(* IEC 61131-3 sources: AXOpen/src/components.abb.robotics/ctrl/src/AxoIrc5_v_1_x_x/TypesStructuresAndEnums, 5 files *)

(* ---- AxoIrc5_v_1_x_x_Component_Status.st ---- *)
NAMESPACE AXOpen.Components.Abb.Robotics
    {S7.extern=ReadWrite}
    {#ix-attr:[Container(Layout.Stack)]}
    CLASS PUBLIC AxoIrc5_v_1_x_x_Component_Status  EXTENDS AXOpen.Components.Robotics.AxoRobot_Status
        VAR PUBLIC
        END_VAR
    END_CLASS
END_NAMESPACE

(* ---- AxoIrc5_v_1_x_x_Config.st ---- *)
NAMESPACE AXOpen.Components.Abb.Robotics
    {#ix-attr:[Container(Layout.Stack)]}
    {S7.extern=ReadWrite}
    CLASS PUBLIC AxoIrc5_v_1_x_x_Config
        VAR PUBLIC
            {#ix-set:AttributeName = "<#Info time#>"}
            InfoTime : LTIME := LT#2S;
            {#ix-set:AttributeName = "<#Error time#>"}
            ErrorTime : LTIME := LT#0S;
            {#ix-set:AttributeName = "<#Task timeout#>"}
            TaskTimeout : LTIME := LT#0S;
            {#ix-set:AttributeName = "<#Hardware IDs#>"}
            HWIDs : AxoIrc5_v_1_x_x_HWIDs;
        END_VAR
    END_CLASS
END_NAMESPACE

(* ---- AxoIrc5_v_1_x_x_Control.st ---- *)
NAMESPACE AXOpen.Components.Abb.Robotics
    {S7.extern=ReadWrite}
    {#ix-attr:[Container(Layout.Wrap)]}
    CLASS AxoIrc5_v_1_x_x_Control
        VAR PUBLIC
            {#ix-attr:[Container(Layout.Stack)]}
            {#ix-attr:[Group(GroupLayout.GroupBox)]}
            {#ix-set:AttributeName = "<#Interuption actually running instruction#>"}
            Interupt : BOOL;
            {#ix-set:AttributeName = "<#Load program#>"}
            LoadProg : BOOL;
            {#ix-set:AttributeName = "<#Load and run program#>"}
            LoadAndStartProg : BOOL;
            {#ix-set:AttributeName = "<#Switch off the motors#>"}
            MotorOff : BOOL;
            {#ix-set:AttributeName = "<#Switch on the motors#>"}
            MotorOn : BOOL;
            {#ix-set:AttributeName = "<#Switch on the motors and start program#>"}
            MotorOnAndStart : BOOL;
            {#ix-set:AttributeName = "<#Emergency stop acknowledge#>"}
            ResetEmgStop : BOOL;
            {#ix-set:AttributeName = "<#Error acknowledge#>"}
            ResetError : BOOL;

            {#ix-attr:[Container(Layout.Stack)]}
            {#ix-attr:[Group(GroupLayout.GroupBox)]}
            {#ix-set:AttributeName = "<#Program start#>"}
            StartProgram : BOOL;
            {#ix-set:AttributeName = "<#Program start at main#>"}
            StartAtMain : BOOL;
            {#ix-set:AttributeName = "<#Program stop#>"}
            StopProgram : BOOL;
            {#ix-set:AttributeName = "<#Stop movement-quick#>"}
            QuickStop : BOOL;
            {#ix-set:AttributeName = "<#Stop movement-soft#>"}
            SoftStop : BOOL;
            {#ix-set:AttributeName = "<#Stop program at the end of the cycle#>"}
            StopCycle : BOOL;
            {#ix-set:AttributeName = "<#Stop program at the end of the instruction#>"}
            StopInstruction : BOOL;
            {#ix-set:AttributeName = "<#Speed limitation#>"}
            LimitSpeed : BOOL;

            {#ix-attr:[Container(Layout.Stack)]}
            {#ix-attr:[Group(GroupLayout.GroupBox)]}
            {#ix-set:AttributeName = "<#Master mode#>"}
            MasterMode : BYTE;

            {#ix-attr:[Container(Layout.Stack)]}
            {#ix-attr:[Group(GroupLayout.GroupBox)]}
            {#ix-set:AttributeName = "<#Tool 1 retract#>"}
            Tool_1_Retract : BOOL;
            {#ix-set:AttributeName = "<#Tool 1 extend#>"}
            Tool_1_Extend : BOOL;
            {#ix-set:AttributeName = "<#Tool 2 retract#>"}
            Tool_2_Retract : BOOL;
            {#ix-set:AttributeName = "<#Tool 2 extend#>"}
            Tool_2_Extend : BOOL;
            {#ix-set:AttributeName = "<#Tool 3 retract#>"}
            Tool_3_Retract : BOOL;
            {#ix-set:AttributeName = "<#Tool 3 extend#>"}
            Tool_3_Extend : BOOL;
            {#ix-set:AttributeName = "<#Tool 4 retract#>"}
            Tool_4_Retract : BOOL;
            {#ix-set:AttributeName = "<#Tool 4 extend#>"}
            Tool_4_Extend : BOOL;

            {#ix-attr:[Container(Layout.Stack)]}
            {#ix-attr:[Group(GroupLayout.GroupBox)]}
            {#ix-set:AttributeName = "<#Zones#>"}
            Zone : BYTE;
            {#ix-set:AttributeName = "<#In position#>"}
            InPosition : BYTE;
            {#ix-set:AttributeName = "<#Action number#>"}
            ActionNo : BYTE;
            {#ix-set:AttributeName = "<#Global robot speed#>"}
            GlobalSpeed : BYTE;
            {#ix-set:AttributeName = "<#Tool number#>"}
            ToolNo : BYTE;
            {#ix-set:AttributeName = "<#Workobject number#>"}
            WorkobjectNo : BYTE;
            {#ix-set:AttributeName = "<#Point number#>"}
            PointNo : BYTE;
            {#ix-set:AttributeName = "<#User specific speed 1#>"}
            UserSpecSpeed1 : REAL;
            {#ix-set:AttributeName = "<#User specific speed 2#>"}
            UserSpecSpeed2 : REAL;

            {#ix-attr:[Container(Layout.Stack)]}
            {#ix-attr:[Group(GroupLayout.GroupBox)]}
            {#ix-set:AttributeName = "<#Coordinates#>"}
            Coordinates : AXOpen.Components.Abstractions.Robotics.AxoRoboticsCoordinates;
        END_VAR
    END_CLASS
END_NAMESPACE

(* ---- AxoIrc5_v_1_x_x_HWIDs.st ---- *)
NAMESPACE AXOpen.Components.Abb.Robotics
{S7.extern=ReadWrite}
CLASS AxoIrc5_v_1_x_x_HWIDs
  VAR PUBLIC
     {#ix-set:AttributeName = "<#Hardware ID of the device#>"}
     HW_Device              :  UINT;
     {#ix-set:AttributeName = "<#Hardware ID of the 'DI_64_bytes' submodule#>"}
     HwID_DI_64_bytes       :   UINT;
     {#ix-set:AttributeName = "<#Hardware ID of the 'DO_64_bytes' submodule#>"}
     HwID_DO_64_bytes          :   UINT;
  END_VAR
END_CLASS
END_NAMESPACE

(* ---- AxoIrc5_v_1_x_x_State.st ---- *)
NAMESPACE AXOpen.Components.Abb.Robotics
    {S7.extern=ReadWrite}
    {#ix-attr:[Container(Layout.Wrap)]}
    CLASS AxoIrc5_v_1_x_x_State
        VAR PUBLIC
            {#ix-attr:[Container(Layout.Stack)]}
            {#ix-attr:[Group(GroupLayout.GroupBox)]}
            {#ix-set:AttributeName = "<#AutoOn#>"}
            AutoOn : BOOL;
            {#ix-set:AttributeName = "<#CycleOn#>"}
            CycleOn : BOOL;
            {#ix-set:AttributeName = "<#Emergency stop#>"}
            EmgStop : BOOL;
            {#ix-set:AttributeName = "<#Error#>"}
            Error : BOOL;
            {#ix-set:AttributeName = "<#Event ID#>"}
            EventId : UDINT;
            {#ix-set:AttributeName = "<#Move active#>"}
            MoveActive : BOOL;
            {#ix-set:AttributeName = "<#Move inactive#>"}
            MoveInactive : BOOL;
            {#ix-set:AttributeName = "<#Motor off#>"}
            MotorOff : BOOL;

            {#ix-attr:[Container(Layout.Stack)]}
            {#ix-attr:[Group(GroupLayout.GroupBox)]}
            {#ix-set:AttributeName = "<#Motor on#>"}
            MotorOn : BOOL;
            {#ix-set:AttributeName = "<#Motor off state#>"}
            MotorOffState : BOOL;
            {#ix-set:AttributeName = "<#Motor on state#>"}
            MotorOnState : BOOL;
            {#ix-set:AttributeName = "<#Program execution error#>"}
            ProgExecError : BOOL;
            {#ix-set:AttributeName = "<#Safety OK#>"}
            SafetyOk : BOOL;
            {#ix-set:AttributeName = "<#System input busy#>"}
            SystemInputBusy : BOOL;
            {#ix-set:AttributeName = "<#Program pointer moved#>"}
            PpMoved : BOOL;
            {#ix-set:AttributeName = "<#Motion supervision#>"}
            MotionSupervision : BOOL;
            {#ix-set:AttributeName = "<#Battery Low#>"}
            BatteryLow : BOOL;

            {#ix-attr:[Container(Layout.Stack)]}
            {#ix-attr:[Group(GroupLayout.GroupBox)]}
            {#ix-set:AttributeName = "<#In area 1#>"}
            InArea_1 : BOOL;
            {#ix-set:AttributeName = "<#In area 2#>"}
            InArea_2 : BOOL;
            {#ix-set:AttributeName = "<#In area 3#>"}
            InArea_3 : BOOL;
            {#ix-set:AttributeName = "<#In area 4#>"}
            InArea_4 : BOOL;
            {#ix-set:AttributeName = "<#In position 1#>"}
            InPosition_1 : BOOL;
            {#ix-set:AttributeName = "<#In position 2#>"}
            InPosition_2 : BOOL;
            {#ix-set:AttributeName = "<#In position 3#>"}
            InPosition_3 : BOOL;
            {#ix-set:AttributeName = "<#In position 4#>"}
            InPosition_4 : BOOL;

            {#ix-attr:[Container(Layout.Stack)]}
            {#ix-attr:[Group(GroupLayout.GroupBox)]}
            {#ix-set:AttributeName = "<#Zones#>"}
            Zone : BYTE;
            {#ix-set:AttributeName = "<#In position#>"}
            InPosition : BYTE;

            {#ix-attr:[Container(Layout.Stack)]}
            {#ix-attr:[Group(GroupLayout.GroupBox)]}
            {#ix-set:AttributeName = "<#Tool 1 retract#>"}
            Tool_1_Retract : BOOL;
            {#ix-set:AttributeName = "<#Tool 1 extend#>"}
            Tool_1_Extend : BOOL;
            {#ix-set:AttributeName = "<#Tool 2 retract#>"}
            Tool_2_Retract : BOOL;
            {#ix-set:AttributeName = "<#Tool 2 extend#>"}
            Tool_2_Extend : BOOL;
            {#ix-set:AttributeName = "<#Tool 3 retract#>"}
            Tool_3_Retract : BOOL;
            {#ix-set:AttributeName = "<#Tool 3 extend#>"}
            Tool_3_Extend : BOOL;
            {#ix-set:AttributeName = "<#Tool 4 retract#>"}
            Tool_4_Retract : BOOL;
            {#ix-set:AttributeName = "<#Tool 4 extend#>"}
            Tool_4_Extend : BOOL;

            {#ix-attr:[Container(Layout.Stack)]}
            {#ix-attr:[Group(GroupLayout.GroupBox)]}
            {#ix-set:AttributeName = "<#Auto stop 1#>"}
            AutoStop_1 : BOOL;
            {#ix-set:AttributeName = "<#Auto stop 2#>"}
            AutoStop_2 : BOOL;
            {#ix-set:AttributeName = "<#Emergency stop 1#>"}
            EmergencyStop_1 : BOOL;
            {#ix-set:AttributeName = "<#Emergency stop 2#>"}
            EmergencyStop_2 : BOOL;
            {#ix-set:AttributeName = "<#General stop 1#>"}
            GeneralStop_1 : BOOL;
            {#ix-set:AttributeName = "<#General stop 2#>"}
            GeneralStop_2 : BOOL;
            {#ix-set:AttributeName = "<#Enable 1#>"}
            Enable_1 : BOOL;
            {#ix-set:AttributeName = "<#Enable 2#>"}
            Enable_2 : BOOL;

            {#ix-attr:[Container(Layout.Stack)]}
            {#ix-attr:[Group(GroupLayout.GroupBox)]}
            {#ix-set:AttributeName = "<#Action number#>"}
            ActionNo : BYTE;
            {#ix-set:AttributeName = "<#Global speed#>"}
            GlobalSpeed : BYTE;
            {#ix-set:AttributeName = "<#Tool number#>"}
            ToolNo : BYTE;
            {#ix-set:AttributeName = "<#Workobject number#>"}
            WorkobjectNo : BYTE;
            {#ix-set:AttributeName = "<#PointNumber#>"}
            PointNo : BYTE;
            {#ix-set:AttributeName = "<#User specific speed 1#>"}
            UserSpecSpeed1 : DINT;
            {#ix-set:AttributeName = "<#User specific speed 2#>"}
            UserSpecSpeed2 : DINT;

            {#ix-attr:[Container(Layout.Stack)]}
            {#ix-attr:[Group(GroupLayout.GroupBox)]}
            {attribute  addProperty Name "<#Coordinates#>"}
            Coordinates : AXOpen.Components.Abstractions.Robotics.AxoRoboticsCoordinates;
        END_VAR
    END_CLASS
END_NAMESPACE
